/// This function block is a container for all axis objects that are used by this unit.
/// The parent of all objects can be directly transfered in their constructor (this is only relevant for equipment objects
/// that have to be managed (e.g. [DebouncedInput](xref:ZEquipment.DebouncedInput), [Light](xref:ZEquipment.Light), ...).
FUNCTION_BLOCK MachineAxis EXTENDS MachineContainer
VAR
  {attribute 'hide'}
  _axisbridge : ZApplication.AxisBridge(_parent);
END_VAR
VAR_INPUT

{attribute '__ZwPlcUnitEquipmentDeclaration__'} // Do not remove this attribute! It is used for code generation.
END_VAR

IF _isInitialized
THEN
  RETURN;
END_IF

  _axisbridge.SetLogger(_parent._logger);

{attribute '__ZwPlcUnitEquipmentImplementation__'} // Do not remove this attribute! It is used for code generation.

_isInitialized := TRUE;

END_FUNCTION_BLOCK

(* stored: Version 1.1.0.1
   POU MachineAxis: Id {0d47c18b-39fd-4f9e-80ae-a66f5d7518df}, SpecialFunc None *)
